Staubli VAL3: default.pjx

Parameters version=s7.7.1 stackSize=5000 millimeterUnit=true
Program file=start.pgx
Program file=stop.pgx
Data file=default.dtx
